# EPICS substitutions: kri_rf/kri_rfApp/Db/kri_rf.substitutions
file kri_rf.template { pattern
{ Sys	, Dev		, PORT		}
{ Depo	, "{RF:1}"	, Depo_RF1	}
}
